FUNCTION_BLOCK ATM_AR_DIVTIME (* Divides a time value by a number value, both via adapters (IN1 as ATM socket instead of a fixed TIME literal, unlike AR_DIVTIME) *)
  (* Standard: 61131-3; Classification: standard arithmetic function; Description: Copyright (c) 2013 TU Wien ACIN This program and the accompanying materials are made available under the terms of the Eclipse Public License 2.0 which is available at https://www.eclipse.org/legal/epl-2.0/ SPDX-License-Identifier: EPL-2.0 *)
  (* Version 3.0, 2025-04-14, Patrick Aigner, changed package *)
  (* Version 1.0, 2013-09-12, Monika Wenger, TU Wien ACIN *)
  PACKAGE adapter::iec61131::arithmetic;
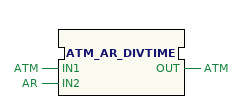
  SOCKETS
    IN1 : adapter::types::unidirectional::ATM; (* Time input to be divided *)
    IN2 : adapter::types::unidirectional::AR; (* Divisor *)
  END_SOCKETS
  PLUGS
    OUT : adapter::types::unidirectional::ATM; (* IN1 divided by IN2 *)
  END_PLUGS
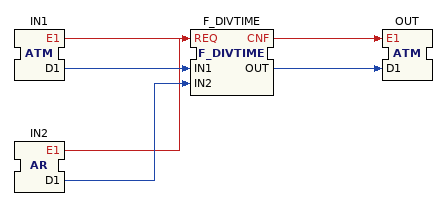
  FBS
    F_DIVTIME : iec61131::arithmetic::F_DIVTIME;
  END_FBS
  EVENT_CONNECTIONS
    F_DIVTIME.CNF TO OUT.E1;
    IN1.E1 TO F_DIVTIME.REQ;
    IN2.E1 TO F_DIVTIME.REQ;
  END_CONNECTIONS
  DATA_CONNECTIONS
    F_DIVTIME.OUT TO OUT.D1;
    IN1.D1 TO F_DIVTIME.IN1;
    IN2.D1 TO F_DIVTIME.IN2;
  END_CONNECTIONS
END_FUNCTION_BLOCK
